ABB RAPID module: Product3Mod.modx

MODULE Product3Mod



    PROC SeqProduct3()
        ProductPick;
        ProductProcess;
        ProductPlace;
    ENDPROC



    LOCAL PROC ProductPick()
        GripClose;
    ENDPROC



    LOCAL PROC ProductProcess()
        !
    ENDPROC



    LOCAL PROC ProductPlace()
        GripOpen;
    ENDPROC



ENDMODULE
